Fanuc KAREL source: kb00021.KL

-- PROVISIONAL review KL for V770-1; original PC SHA256 7fa497a5b03df607b727b5d1d81c7b99996c8b530589cc1568c5c4969c7049f2
-- Incomplete behavior may be omitted. Consult companion uncertainty JSON. Do not deploy.
PROGRAM KB00021
%NOLOCKGROUP
BEGIN
  -- UNRESOLVED_PC offsets 5-14; opcodes 3F,75
  -- UNRESOLVED_PC offsets 19-26; opcodes 9D,23
  -- UNRESOLVED_PC offsets 31-49; opcodes 27,22,2A,22,31
  -- UNRESOLVED_PC offsets 54-58; opcodes 7F
END KB00021
